FUNCTION_BLOCK Test_WhenBusy_SetDone_SetsDone EXTENDS TUnitTestbase
VAR
END_VAR

METHOD  Execute
VAR_INST
    Execution : TExecution;
END_VAR
Test_Started();

Execution.Start();
Execution.SetBusy();
Execution.SetDone();

Assertion.AssertEquals_BOOL(
    Expected := TRUE,
    Actual   := Execution.Done,
    ObjectName := _TestName,
    VariableName  := 'Execution.Done');

Assertion.AssertEquals_BOOL(
    Expected := TRUE,
    Actual   := Execution.Ready,
    ObjectName := _TestName,
    VariableName  := 'Execution.Ready');

Test_Finished();
END_METHOD

END_FUNCTION_BLOCK

(* stored: Version 1.1.0.1, ProductVersion 3.1.4024.3
   POU Test_WhenBusy_SetDone_SetsDone: Id {0711fba5-2047-4dd9-974b-a4271be3afd0}, SpecialFunc None
   Method Execute: Id {5bb87ee5-d21b-4074-aa65-95dc1ff4aebd} *)
